# EPICS autosave request: iocBoot/gmca_23b_ioc2/dbSave/KB_Hy_.req
%
% BURT Request File
%
% $(P)KB:Hy:  Horizontal KB mirror Y-positioning
%

file assy.req ASSY=$(P)KB:Hy
$(P)KB:Hy:BaseLength
file mtr1.req MTR1=$(P)KB:mhy1
file mtr1.req MTR1=$(P)KB:mhy2
file drv1.req DRV1=$(P)KB:HY1
file drv1.req DRV1=$(P)KB:HY2
file axs1.req AXS1=$(P)KB:HY
file axs1.req AXS1=$(P)KB:HA
